Yaskawa INFORM job: VAN-ONDER-NAAR-BOVEN.JBI

/JOB
//NAME VAN-ONDER-NAAR-BOVEN
//POS
///NPOS 5,0,0,0,0,0
///TOOL 1
///POSTYPE PULSE
///PULSE
C00000=9246,34629,-214651,-6202,174139,325719
C00001=9246,-64041,-214651,-6202,174139,325719
C00002=9246,-89754,-52204,-6202,55462,325719
C00003=9246,-89754,67013,-6202,-162538,32377
C00004=-5869,-28950,85500,-7487,-122252,35389
//INST
///DATE 2025/03/05 16:07
///ATTR SC,RW
///GROUP1 RB1
NOP
MOVJ C00000 VJ=100.00
MOVJ C00001 VJ=100.00
MOVJ C00002 VJ=100.00
MOVJ C00003 VJ=100.00
MOVJ C00004 VJ=100.00
END
